// TIA Portal V20 export
VAR_GLOBAL   // PLC tag table "cmd_Robot"
END_VAR
VAR_GLOBAL CONSTANT   // user constants
   CMD_RobotChangeDataForGripper : Int := 10;
   CMD_RobotPickGripper : Int := 11;
   CMD_RobotRemoveGripper : Int := 12;
   CMD_RobotPickObject : Int := 13;
   CMD_RobotPlaceObject : Int := 14;
   CMD_RobotPositioning : Int := 15;
   CMD_RobotPickPlaceObject : Int := 16;
   CMD_RobotToHomePos : Int := 20;
   CMD_RobotMaintenancePos : Int := 21;
   CMD_RobotRemoteMode : Int := 81;
   CMD_RobotLocalMode : Int := 82;
   CMD_RobotResetObjectOnGripper : Int := 83;
   CMD_RobotReset : Int := 99;
   CMD_RobotExtractTray : Int := 25;
   CMD_RobotReleaseTray : Int := 26;
   CMD_RobotPositioning_MC1 : Int := 1511;
   CMD_RobotPositioning_MC2 : Int := 1512;
   CMD_RobotPositioning_BOX1 : Int := 1501;
   CMD_RobotPositioning_BOX2 : Int := 1502;
   CMD_HOLD : Int := 17;
   PosROBOT : Int := 1000;   // codice della posizione della flangia robot
   CMD_RestartMainProg : Int := 18;
   CMD_changeRobotSpeed : Int := 100;
   CMD_RobotSwapGripper : Int := 30;
   CMD_HMI_SwapGripper : Int := 27;
   CMD_RobotPickPartTray : Int := 31;
   CMD_RobotPlacePartTray : Int := 32;
   CMD_RobotPickPartMC : Int := 33;
   CMD_RobotPlacePartMC : Int := 34;
   CMD_DeclarePallet_MC : Int := 40;
   CMD_RemovePallet_MC : Int := 41;
   CMD_ManualViceOn : Int := 42;
   CMD_ManualViceOff : Int := 43;
   CMD_Refresh : Int := 90;
   CMD_RobotDeclareState : Int := 35;
   _Declare_State : Int := 31;
   CMD_OpenGripper1 : Int := 240;
   CMD_CloseGripper1 : Int := 241;
   CMD_OpenGripper2 : Int := 242;
   CMD_CloseGripper2 : Int := 243;
   CMD_RobotOpenGripper1 : Int := 1;
   CMD_RobotCloseGripper1 : Int := 2;
   CMD_RobotOpenGripper2 : Int := 3;
   CMD_RobotCloseGripper2 : Int := 4;
   CMD_RobotPickPlacePartMC : Int := 244;
   CMD_DeclarePiece_MC : Int := 36;
   CMD_RemovePiece_MC : Int := 37;
   CMD_DeclareTray_BOX : Int := 38;
   CMD_DeclarePosition_TRAY : Int := 39;
   CMD_DeclarePieceType_TRAY : Int := 44;
END_VAR
